(* CoDeSys 2.3.9.28 project: CSV_Config.pro *)
(* Libraries: SysLibFile.lib 2.12.10 05:48:34, Standard.lib 2.12.10 05:48:34, SYSLIBCALLBACK.LIB 2.12.10 05:48:32 *)

(* PLC configuration (modules and I/O channels)
AT %IB0 [BYTEOnB_I] First Byte of 8
AT %QB0 [BYTEOnB_Q] First Byte of 8
Fieldbus variables [FB_VARS] node 1, in %IB512 out %QB512
*)

(* Task configuration *)
TASK Sampling (PRIORITY := 1, INTERVAL := T#200ms);
	PLC_PRG();
END_TASK

(* Global variable list: Globale_Variablen *)
VAR_GLOBAL CONSTANT
	iMaxParams			:INT:=5;(* Number of Parameters per File *)
	gc_ParameterCount	:INT:=1;(* Number of Values per Parameter *)
	gc_RawDataSize		:UINT:=500; (* Raw data size for reading in file ASCII *)
END_VAR

(* Data type *)
TYPE typCSV :
STRUCT
	sDescription	:STRING;
	Parameter		:ARRAY[1..gc_ParameterCount] OF REAL;
END_STRUCT
END_TYPE

(* POU PLC_PRG, FBD *)
PROGRAM PLC_PRG
(*
  Function: 	Reading a CSV file
  Description: 	This project shows a functionblock which reads data from a CSV file into an array.
				Each line in the CSV contains a description and a real value.
				Each parameter  is terminated by CR LF.

---- Example CSV File -----

A_Value;245345
B_Value;0							
C_Value;8.3							
D_Value;-123439.3 						
E_Value;1						*)

VAR
	xLoad			: BOOL; (* Initiate load operation *)
	xSave			: BOOL; (* Initiate save operation *)
	sLoadStatus		: STRING; (* Feedback on load *)
	sSaveStatus		: STRING; (* Feedback on save *)
	ConfigData		: ARRAY [1..iMaxParams] OF  typCSV; (* Structure with the config data being loaded or saved *)
	sFileName		: STRING := 'config.csv'; (* Working Filename *)
	bSeperator 		: BYTE := 59; (* Semicolon (;) is the seperator between parameter and value. *)
	iError			: INT; (* Error Code for Save *)
	xWriteToSD		: BOOL; (* User selectable location for file operation, on = 750-880 SD, off = internal flash *)
	sFilePath		: STRING; (* SD card is S:\, Internal Path is blank, but this points to the PLC folder *)
	sFilePath_Name	: STRING; (* Complete path + filename *)
END_VAR
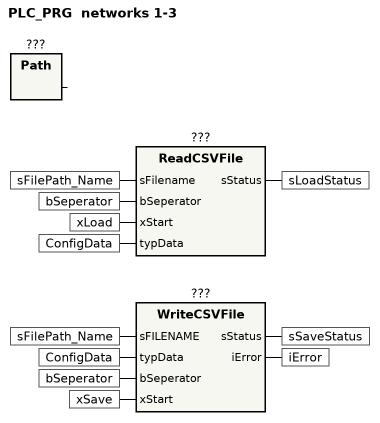
_FBD_ (* Function Block Diagram *)
NETWORK 1
	???:Path()
NETWORK 2
	???:ReadCSVFile(sFilename: sFilePath_Name, bSeperator: bSeperator, xStart: xLoad, typData: ConfigData) => sLoadStatus
NETWORK 3
	???:WriteCSVFile(sFILENAME: sFilePath_Name, typData: ConfigData, bSeperator: bSeperator, xStart: xSave, iError => iError) => sSaveStatus
_END_FBD_
END_PROGRAM
ACTION Path:
IF xWriteToSD THEN
	sFilePath := 'S:\';
ELSE
	sFilePath := '';
END_IF
sFilePath_Name := CONCAT(sFilePath, sFileName);
END_ACTION

(* POU ReadCSVFile, ST *)
PROGRAM ReadCSVFile
VAR_INPUT
	sFilename		:STRING;
	bSeperator		:BYTE:=59;(*seperator semicolon:59=;*)
END_VAR
VAR_IN_OUT
	xStart			:BOOL;
	typData			:ARRAY [1..iMaxParams] OF  typCSV;
END_VAR
VAR_OUTPUT
	sStatus			:STRING;
END_VAR
VAR
	bEndOfFile		:BYTE:=13;
	FileIdent		:DWORD;
	rawdata			:ARRAY[0..gc_RawDataSize] OF BYTE;
	filesizev		:DINT;
	tempstring		:STRING;
	startposition	:INT;
	i				:INT;
	j				:INT;
	k				:INT;
END_VAR
IF xStart THEN
	FileIdent:=SysFileOpen(FileName:=sFilename, Mode:='r');
	IF fileident<>0 THEN
		SysFileRead(File:=Fileident, Buffer:=ADR(rawdata), Size:=SIZEOF(rawdata));
		filesizev:=SysFileGetSize(FileName:=sFilename);
		IF filesizev>gc_RawDataSize THEN
			filesizev:=gc_RawDataSize;
		END_IF
		SysFileClose(File:=fileident);(*this function is blocking*)
	ELSE
		sStatus:='File does not exist';
		xStart:=FALSE;
		RETURN;(*no such file available*)
	END_IF
(*copy data to typData array*)
	startposition:=0;
	i:=0;
	FOR j:=1 TO iMaxParams DO
		(*First value in dataset is of type DT. The following value is seperated by bSeperator*)
		WHILE rawdata[startposition+i]<>bSeperator DO
			i:=i+1;
		END_WHILE
		rawdata[startposition+i]:=0;
		MEMCPY(pSourceAddress:=ADR(rawdata[startposition]), pDestinationAddress:=ADR(tempstring), BytesToCopy:=i+1);
		typdata[j].sDescription:=tempstring;
		startposition:=startposition+i+1;
		i:=0;
		(*The parameter values are of type word. The following values are seperated by bSeperator*)
		FOR k:=1 TO gc_ParameterCount-1 DO
			WHILE rawdata[startposition+i]<>bSeperator DO
				i:=i+1;
			END_WHILE
			rawdata[startposition+i]:=0;
			MEMCPY(pSourceAddress:=ADR(rawdata[startposition]), pDestinationAddress:=ADR(tempstring), BytesToCopy:=i+1);
			typdata[j].Parameter[k]:=STRING_TO_REAL(tempstring);
			startposition:=startposition+i+1;
			i:=0;
		END_FOR
		(*Copying the last parameter from typ word. The data set is terminated by CR LF*)
		WHILE rawdata[startposition+i]<>bEndOfFile DO
			i:=i+1;
		END_WHILE
		rawdata[startposition+i]:=0;
		MEMCPY(pSourceAddress:=ADR(rawdata[startposition]), pDestinationAddress:=ADR(tempstring), BytesToCopy:=i+1);
		typdata[j].Parameter[k]:=STRING_TO_REAL(tempstring);
		startposition:=startposition+i+2;(*The data set is terminated by CR LF(13,10)*)
		i:=0;
	END_FOR
(*copy data to typData array finished*)
	sStatus:='Data read OK';
	xStart:=FALSE;
END_IF
END_PROGRAM

(* POU MEMCPY, ST *)
(*---------------------------------------------------------------------------------------
  WAGO Kontakttechnik GmbH Hansastr. 27 32423 Minden(Westf.) 
  Tel. +49571/887-0 Fax. +49571/887-0                
                                                                                                
  Project: IEC1131 internal library
  
  Function: MEMCPY
  Description: This function copies BytesToCopy bytes from the source
                         address pSourceAddress to the destination address
                         pDestinationAddress
  Date: 25.09.2000

------------------------------------------------------------------------------------------*)
FUNCTION MEMCPY:BOOL
VAR_INPUT
	pSourceAddress:							POINTER TO ARRAY[1..2] OF BYTE;
	pDestinationAddress:						POINTER TO ARRAY[1..2] OF BYTE;
	BytesToCopy:								DINT;
END_VAR
VAR
END_VAR
WHILE (BytesToCopy > 0) DO
	pDestinationAddress^[1]:=pSourceAddress^[1]; (* copy bytes from source to destination *)
	pDestinationAddress:=ADR(pDestinationAddress^[2]); (* increment destination *)
	pSourceAddress:=ADR(pSourceAddress^[2]);(* increment source *)
	BytesToCopy:=BytesToCopy -1; (* decrement number of bytes to copy *)
END_WHILE
END_FUNCTION

(* POU WriteCSVFile, ST *)
PROGRAM WriteCSVFile
(* 	This function block Writes the contents of the data structure to a CSV File

	Required Libraries:
		Standard.lib
		SysLibFile.lib
*)
VAR_INPUT
	sFILENAME 		:STRING(80); (* Filename to store data to (e.g. 'config.csv' 		*)
	typData			:ARRAY [1..iMaxParams] OF typCSV;
	bSeperator		:BYTE :=59;	(* Seperator semicolon:59=;*)
END_VAR
VAR_IN_OUT
	xStart 			:BOOL;	(* Set TRUE to write data, set False to stop.		 *)
END_VAR
VAR_OUTPUT
	sStatus			:STRING;
	iError 			:INT;	(* 00 : Normal Operation	*)
							(* 90 : Can't Open File 	*)
							(* 91 : Can't Close File 	*)
							(* 92 : Can't Write to File 	*)
END_VAR
VAR
	FileOpen		:BOOL := FALSE;
	handle			:DWORD;
	Mode			:STRING[20] := 'rw'; (* read/write *)
	DataString 		:STRING(80);
	i				:INT;
END_VAR
IF xStart THEN
	sStatus := 'Try to open file';
	IF NOT FileOpen THEN
		(* Open File *)
		handle := SysFileOpen(sFileName, Mode);
		IF handle > 0 THEN
			FileOpen := TRUE;
			sStatus := 'File Open OK.';
		ELSE
			iERROR := 90; (* Could not open file. *)
			sStatus := 'Could not open file.';
		END_IF
	END_IF
	
	IF FileOpen THEN
		FOR i := 1 TO iMaxParams DO
				DataString := TypData[i].sDescription;
				DataString := CONCAT(DataString,ASCIIBYTE_TO_STRING(bSeperator));
				DataString := CONCAT(DataString,REAL_TO_STRING(TypData[i].Parameter[1]));
	
				DataString := CONCAT(DataString,ASCIIBYTE_TO_STRING(13)); (* CR *)
				DataString := CONCAT(DataString,ASCIIBYTE_TO_STRING(10)); (* LF *)
				(* Write string to file *)
				IF SysFileWrite(handle, ADR(DataString), LEN(DataString)) = 0 THEN
					iERROR := 92; (* Could not write to file *)
					sStatus := 'Could not write file.';
				END_IF
		END_FOR
	END_IF
	
	IF FileOpen THEN
		(* Close file *)
		IF SysFileClose(handle) THEN
			FileOpen := FALSE;
			sStatus := 'File Saved.';
		ELSE
			iERROR := 91; (* Could not close file *)
			sStatus := 'Could not close file.';
		END_IF
		xStart := FALSE;
	END_IF
END_IF
END_PROGRAM

(* Visualisation PLC_VISU
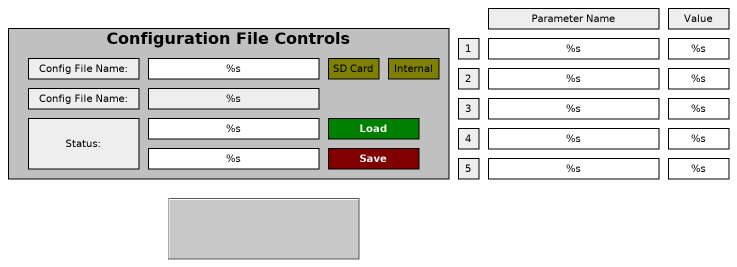
rectangle at (20,50)-(461,201): text "Configuration File Controls"
rectangle at (340,140)-(431,161): text "Load"; alarm colour if PLC_PRG.xLoad; toggles PLC_PRG.xLoad
rectangle at (40,80)-(151,101): text "Config File Name:"
rectangle at (160,80)-(331,101): text "%s"; shows PLC_PRG.sFileName; editable
rectangle at (40,140)-(151,191): text "Status:"
rectangle at (160,140)-(331,161): text "%s"; shows PLC_PRG.sLoadStatus
rectangle at (500,30)-(671,51): text "Parameter Name"
rectangle at (500,60)-(671,81): text "%s"; shows PLC_PRG.ConfigData[1].sDescription; editable
rectangle at (680,30)-(741,51): text "Value"
rectangle at (680,60)-(741,81): text "%s"; shows PLC_PRG.ConfigData[1].Parameter[1]; editable
rectangle at (470,60)-(491,81): text "1"
rectangle at (500,90)-(671,111): text "%s"; shows PLC_PRG.ConfigData[2].sDescription; editable
rectangle at (680,90)-(741,111): text "%s"; shows PLC_PRG.ConfigData[2].Parameter[1]; editable
rectangle at (470,90)-(491,111): text "2"
rectangle at (500,120)-(671,141): text "%s"; shows PLC_PRG.ConfigData[3].sDescription; editable
rectangle at (680,120)-(741,141): text "%s"; shows PLC_PRG.ConfigData[3].Parameter[1]; editable
rectangle at (470,120)-(491,141): text "3"
rectangle at (500,150)-(671,171): text "%s"; shows PLC_PRG.ConfigData[4].sDescription; editable
rectangle at (680,150)-(741,171): text "%s"; shows PLC_PRG.ConfigData[4].Parameter[1]; editable
rectangle at (470,150)-(491,171): text "4"
rectangle at (500,180)-(671,201): text "%s"; shows PLC_PRG.ConfigData[5].sDescription; editable
rectangle at (680,180)-(741,201): text "%s"; shows PLC_PRG.ConfigData[5].Parameter[1]; editable
rectangle at (470,180)-(491,201): text "5"
rectangle at (340,170)-(431,191): text "Save"; alarm colour if PLC_PRG.xSave; toggles PLC_PRG.xSave
rectangle at (160,170)-(331,191): text "%s"; shows PLC_PRG.sSaveStatus
rectangle at (340,80)-(391,101): text "SD Card"; alarm colour if PLC_PRG.xWriteToSD; toggles PLC_PRG.xWriteToSD
rectangle at (400,80)-(451,101): text "Internal"; alarm colour if NOT PLC_PRG.xWriteToSD; toggles PLC_PRG.xWriteToSD
rectangle at (40,110)-(151,131): text "Config File Name:"
rectangle at (160,110)-(331,131): text "%s"; shows PLC_PRG.sFilePath_Name
1 more shapes without text or variables
*)
